// TIA Portal V17 export
// export: Created 2022-10-14T12:26:28.8296594Z, ExportSetting WithDefaults, DisplayName Totally Integrated Automation Portal, DisplayVersion V17 Update 4, DisplayName TIA Portal Openness, DisplayVersion V17 Update 4, DisplayName TIA Portal Version Control Interface, DisplayVersion V17, DisplayName SINAMICS Startdrive Advanced, DisplayVersion V17 Update2, DisplayName SINAMICS Startdrive G130, G150, S120, S150, SINAMICS MV, S210, DisplayVersion V17 Update2, DisplayName SINAMICS Startdrive G110M, G120, G120C, G120D, G120P, G115D, DisplayVersion V17 Update2, DisplayName STEP 7 Professional, DisplayVersion V17 Update 4, DisplayName STEP 7 Safety, DisplayVersion V17, DisplayName WinCC Advanced / Unified PC, DisplayVersion V17 Update 4
FUNCTION "Kreis_AWL" : Void   // FC3, STL
{ S7_Optimized_Access := 'TRUE' }
VERSION : 0.1
// stored: AutoNumber true, UDAEnableTagReadback false
   VAR_INPUT
      INput_INT : Int;
      INput_MAX_INT : Int;
      X0_POS : Int;
      Y0_POS : Int;
      Anfang_Grad : Real;   // Startwinkel
      Radius : Real;
      Clockwise : Bool;   // Im Uhrzeigersinn / Gegen den Uhrzeigersinn
   END_VAR
   VAR_OUTPUT
      X_POS : Int;   // verbinden mit HMI
      Y_POS : Int;   // verbinden mit HMI
   END_VAR
   VAR_TEMP
      Bodenmass : Real;
      Grad_per_input : Real;
      Richtung : Real;
   END_VAR
BEGIN

NETWORK
TITLE = 
// mit dieser Funktion können Objekte auf einer kreisbahn verschoben werden
      L     360.0;
      L     #INput_MAX_INT;
      ITD;
      DTR;
      /R;
      T     #Grad_per_input;
//==============================================
      A     #Clockwise;
      JC    m01;
      L     -1.0;
      T     #Richtung;
m01:  NOP   0;
      A     #Clockwise;
      JCN   m02;
      L     1.0;
      T     #Richtung;
m02:  NOP   0;
//=================================================
      L     #INput_INT;
      ITD;
      DTR;
      L     #Grad_per_input;
      *R;
      L     #Anfang_Grad;
      +R;
      L     3.1428;
      *R;
      L     180.0;
      /R;
      L     #Richtung;
      *R;
      T     #Bodenmass;
//======================================================
      L     #Bodenmass;
      COS;
      L     #Radius;
      *R;
      TRUNC;
      L     #X0_POS;
      +I;
      T     #X_POS;
//==================================================
      L     #Bodenmass;
      SIN;
      L     #Radius;
      *R;
      TRUNC;
      L     #Y0_POS;
      +I;
      T     #Y_POS;
//===================================================================


END_FUNCTION
